Staubli VAL3: onF7Event.pgx

program onF7Event()
  local string l_sMessage
  local bool l_bContinue
  local bool l_bYes
  local string l_sItem
  local bool l_bInside
begin
  // look if the bButton is enable
  if bButton[6]
    //
    // STOP /START
    //
    if !cycleStatus:bSimulation and nKey!=255
      if nPoint!=0
        // not for the first point
        call isAtPoint(nPoint,l_bInside)
      else
        l_bInside=true
      endIf
      if l_bInside
        // START
        bStepping=false
        call startCycle(nPoint)
      else
        // not at point
        call language:message(l_sMessage,95)
        call use:timerDialog(l_sMessage+toString("",nPoint+1),2)
      endIf
    elseIf cycleStatus:bSimulation
      // STOP CYCLE
      call stopCycle()
      call use:nullKey(nKey)
    endIf
    //
    //
    use:bUseRefresh=true
    //
  endIf
end
